// TIA Portal V19 export
VAR_GLOBAL   // PLC tag table "AIN"
END_VAR
